{attribute 'GeneratedUsingTerminal: EK1122-0000-0018'}
{attribute addProperty BoxType "EK1122-0000-0018"}
{attribute addProperty Id "Term_153_EK1100Term_153_EK1100_91C0BB4862Term_178_EK1100Term_178_EK1100_9B7E985262"}
{attribute addProperty CRC "3395968278"}
{attribute addProperty Size "124"}
{attribute addProperty Name "Term 147 (EK1122)"}
TYPE Term_147_EK1122_CA6A5D16 EXTENDS EK1122_1FC0878B :
STRUCT
	{attribute addProperty Name "Term 153 (EK1100)"}
	{attribute addProperty PreviousPort "Term 147 (EK1122) : D"}
	{attribute addProperty SyncUnit "default"}
	Term_153_EK1100 : Term_153_EK1100_91C0BB48;
	{attribute addProperty Name "Term 178 (EK1100)"}
	{attribute addProperty PreviousPort "Term 147 (EK1122) : B"}
	{attribute addProperty SyncUnit "default"}
	Term_178_EK1100 : Term_178_EK1100_9B7E9852;
END_STRUCT
END_TYPE

(* stored: Version 1.2.0.0, ProductVersion 3.1.4024.11
   DUT Term_147_EK1122_CA6A5D16: Id {762e7a1f-058e-03b0-2ee6-f3be8c23e369} *)
